TYPE TcoStruct :
STRUCT
	Parent : ITcoObject;
END_STRUCT
END_TYPE

(* stored: Version 1.1.0.1
   DUT TcoStruct: Id {ed0cd97c-0c84-053d-1273-5475387e48d0} *)
